// Mitsubishi GX Works2 project: Pneumalektro   PLC: Q00J

// global labels: Global1
VAR_GLOBAL
  Kör AT X0 : BOOL;
  Kap_1 AT X1 : BOOL;
  Steg_1 AT M0 : BOOL;
  Po_Min AT X2 : BOOL;
  Vrid_Min AT X10 : BOOL;
  Cyl1 AT X7 : BOOL;
  Steg_2 AT M1 : BOOL;
  Stopp AT X15 : BOOL;
  Reset AT X1 : BOOL;
  Magasin AT X2 : BOOL;
  Mag1 : BOOL;
  VitKnapp AT X3 : BOOL;
  MetallKnapp AT X4 : BOOL;
  SvartKnapp AT X5 : BOOL;
  Till_Lager1 : BOOL;
  Till_Lager2 : BOOL;
  Till_Lager3 : BOOL;
  Till_Band : BOOL;
  Hämta : BOOL;
  Cyl1Ute AT X7 : BOOL;
END_VAR

// task Task_01 (event TRUE, interval 0, priority 31): Sekvens, Activation

PROGRAM Sekvens
VAR
  På : BOOL;
  Indu : BOOL;
  Kap : BOOL;
  OK_to_RUN : BOOL;
  Photo : BOOL;
  Metall : BOOL;
  Vit : BOOL;
  Svart : BOOL;
  Reset : BOOL;
  MetallUt : BOOL;
  VitUt : BOOL;
  SvartUt : BOOL;
  Till_Lager : BOOL;
END_VAR
(* structured ladder/FBD written out as ST: instructions are called as NAME(EN, inputs, outputs); _pN, _eN, _tN stand for wires *)
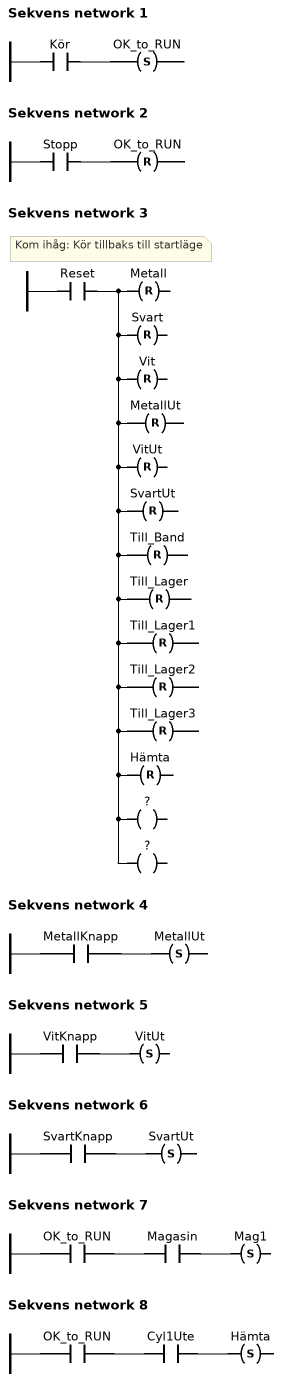
(* network 1 OkToRun *)
SET(Kör, OK_to_RUN);
(* network 2 !OkToRun *)
RST(Stopp, OK_to_RUN);
(* network 3 Reset *)
(* Kom ihåg: Kör tillbaks till startläge *)
RST(Reset, Metall);
RST(Reset, Svart);
RST(Reset, Vit);
RST(Reset, MetallUt);
RST(Reset, VitUt);
RST(Reset, SvartUt);
RST(Reset, Till_Band);
RST(Reset, Till_Lager);
RST(Reset, Till_Lager1);
RST(Reset, Till_Lager2);
RST(Reset, Till_Lager3);
RST(Reset, Hämta);
? := Reset;
? := Reset;
(* network 4 Val Met *)
SET(MetallKnapp, MetallUt);
(* network 5 Val Vit *)
SET(VitKnapp, VitUt);
(* network 6 Val Sva *)
SET(SvartKnapp, SvartUt);
(* network 7 Mag? *)
SET(OK_to_RUN AND Magasin, Mag1);
(* network 8 Hämta? *)
SET(OK_to_RUN AND Cyl1Ute, Hämta);
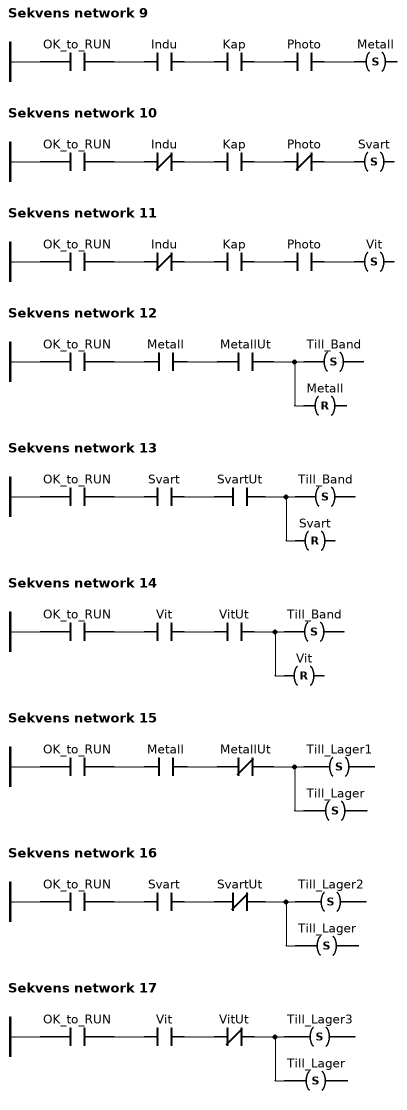
(* network 9 Metall? *)
SET(OK_to_RUN AND Indu AND Kap AND Photo, Metall);
(* network 10 Svart? *)
SET(OK_to_RUN AND NOT Indu AND Kap AND NOT Photo, Svart);
(* network 11 Vit? *)
SET(OK_to_RUN AND NOT Indu AND Kap AND Photo, Vit);
(* network 12 TillBand *)
_p1 := OK_to_RUN AND Metall AND MetallUt;
SET(_p1, Till_Band);
RST(_p1, Metall);
(* network 13 TillBand *)
_p1 := OK_to_RUN AND Svart AND SvartUt;
SET(_p1, Till_Band);
RST(_p1, Svart);
(* network 14 TillBand *)
_p1 := OK_to_RUN AND Vit AND VitUt;
SET(_p1, Till_Band);
RST(_p1, Vit);
(* network 15 ToLager *)
_p1 := OK_to_RUN AND Metall AND NOT MetallUt;
SET(_p1, Till_Lager1);
SET(_p1, Till_Lager);
(* network 16 ToLager *)
_p1 := OK_to_RUN AND Svart AND NOT SvartUt;
SET(_p1, Till_Lager2);
SET(_p1, Till_Lager);
(* network 17 ToLager *)
_p1 := OK_to_RUN AND Vit AND NOT VitUt;
SET(_p1, Till_Lager3);
SET(_p1, Till_Lager);
END_PROGRAM

PROGRAM Activation
END_PROGRAM
